Omron Sysmac Studio project OSU_Capstone_PI_Control (Sysmac Studio 1.47.0.64008, StandardProject)

# Controller new_Controller_0: NX1P2-9024DT1 version 1.40
Units and slaves: Unit 1 : NX-CIF101 (N1)
Task PrimaryTask (priority 4, period or condition 2000): Program0

VAR_GLOBAL
    Goto_Position : REAL := 0.0;
END_VAR
VAR_GLOBAL CONSTANT
    N1_Node_location_information : _sNXUNIT_ID := (NodeAdr := 65535, IPAdr := [5(16#FF)], UnitNo := 1, Path := [16#1, 16#0, 16#2, 16#0, 16#1, 59(16#0)], PathLength := 6);
END_VAR
VAR_GLOBAL
    DevicePort : _sDEVICE_PORT;
    trigger : BOOL;
    SendCfg : _sSERIAL_CFG;
    SendDat : ARRAY[0..49] OF BYTE;
    SendSiz : UINT;
    NX_SerialSend_FB_done : BOOL;
    NX_SerialSend_FB_busy : BOOL;
    NX_SerialSend_FB_err : BOOL;
    NX_SerialSend_FB_errID : WORD;
    trigger1 : BOOL;
    RecvCfg : _sSERIAL_CFG;
    RecvOption : _sSERIAL_RCV_OPTION;
    NX_SerialRcv_FB_done : BOOL;
    RecvDat : ARRAY[0..254] OF BYTE;
    NX_SerialRcv_FB_busy : BOOL;
    NX_SerialRcv_FB_err : BOOL;
    NX_SerialRcv_FB_errID : WORD;
    RecvSize : UINT;
    RecvStringDat : STRING[256];
    restarting : BOOL;
    N1_Ch1_Input_SID : USINT;  (* at IOBus://unit#1/Ch1 Input SID *)
    N1_Ch1_Output_SID_Response : USINT;  (* at IOBus://unit#1/Ch1 Output SID Response *)
    N1_Ch1_Input_Sub_Info : WORD;  (* at IOBus://unit#1/Ch1 Input Sub Info *)
    N1_Ch1_Receive_Command_Flag : BOOL;  (* at IOBus://unit#1/Ch1 Input Data Type/Ch1 Receive Command Flag *)
    N1_Ch1_Send_Command_Flag : BOOL;  (* at IOBus://unit#1/Ch1 Output Data Type/Ch1 Send Command Flag *)
    Pos_String : STRING[15];
    E001_Output_Data_1 : DINT;  (* at ECAT://node#1/Output Data 1 *)
    E001_READY : BOOL;  (* at ECAT://node#1/Sensor Head Status Signal1/READY *)
    E001_STABILITY : BOOL;  (* at ECAT://node#1/Sensor Head Status Signal2/STABILITY *)
END_VAR

PROGRAM Program0
VAR
    NX_SerialSend_FB : NX_SerialSend;
    NX_SerialRcv_FB : NX_SerialRcv;
    clear_trigger : BOOL;
    CmdStage : INT;
    CIFCmdCode : WORD;
    ExpectedOutputSIDResponse : USINT;
    Servo_On : BOOL;
    Reference : BOOL;
    Move_Axis : BOOL;
    Get_Info : BOOL;
    Abort_Send : BOOL;
    Reset_Error : BOOL;
    Pos_length : UINT;
    Last_positon : REAL;
    Auto : BOOL;
    Run : BOOL;
    Next_Move : TON;
    Next_Pos : BOOL;
    ZW_Real : REAL;
    ZW_Temp : REAL;
END_VAR
VAR_EXTERNAL
    DevicePort : _sDEVICE_PORT;
END_VAR
VAR_EXTERNAL CONSTANT
    N1_Node_location_information : _sNXUNIT_ID;
END_VAR
VAR_EXTERNAL
    trigger : BOOL;
    SendCfg : _sSERIAL_CFG;
    SendDat : ARRAY[0..49] OF BYTE;
    SendSiz : UINT;
    NX_SerialSend_FB_done : BOOL;
    NX_SerialSend_FB_busy : BOOL;
    NX_SerialSend_FB_err : BOOL;
    NX_SerialSend_FB_errID : WORD;
    trigger1 : BOOL;
    RecvCfg : _sSERIAL_CFG;
    RecvOption : _sSERIAL_RCV_OPTION;
    NX_SerialRcv_FB_done : BOOL;
    RecvDat : ARRAY[0..254] OF BYTE;
    NX_SerialRcv_FB_busy : BOOL;
    NX_SerialRcv_FB_err : BOOL;
    NX_SerialRcv_FB_errID : WORD;
    RecvSize : UINT;
    RecvStringDat : STRING[256];
    N1_Ch1_Input_SID : USINT;
    N1_Ch1_Output_SID_Response : USINT;
    restarting : BOOL;
    N1_Ch1_Send_Command_Flag : BOOL;
    N1_Ch1_Receive_Command_Flag : BOOL;
    N1_Ch1_Input_Sub_Info : WORD;
    Goto_Position : REAL;
    Pos_String : STRING[15];
    E001_STABILITY : BOOL;
    E001_READY : BOOL;
    E001_Output_Data_1 : DINT;
END_VAR
VAR
    _e1 : R_TRIG;
    _e2 : R_TRIG;
    _e3 : R_TRIG;
    _e4 : R_TRIG;
    _e5 : R_TRIG;
    _e6 : R_TRIG;
    _e7 : R_TRIG;
    _e8 : R_TRIG;
    _e9 : R_TRIG;
END_VAR

(* Section Serial_Setup: ladder, written here as Structured Text *)

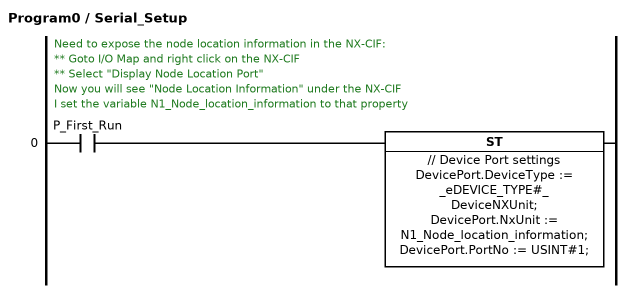
(* Rung 0: Need to expose the node location information in the NX-CIF: / ** Goto I/O Map and right click on the NX-CIF / ** Select "Display Node Location Port" / Now you will see "Node Location Information" under the NX-CIF / I set the variable N1_Node_location_information to that property *)
IF P_First_Run THEN
    // Device Port settings
    DevicePort.DeviceType := _eDEVICE_TYPE#_DeviceNXUnit;
    DevicePort.NxUnit := N1_Node_location_information;
    DevicePort.PortNo := USINT#1;
END_IF;

(* Section Serial_Send: ladder, written here as Structured Text *)

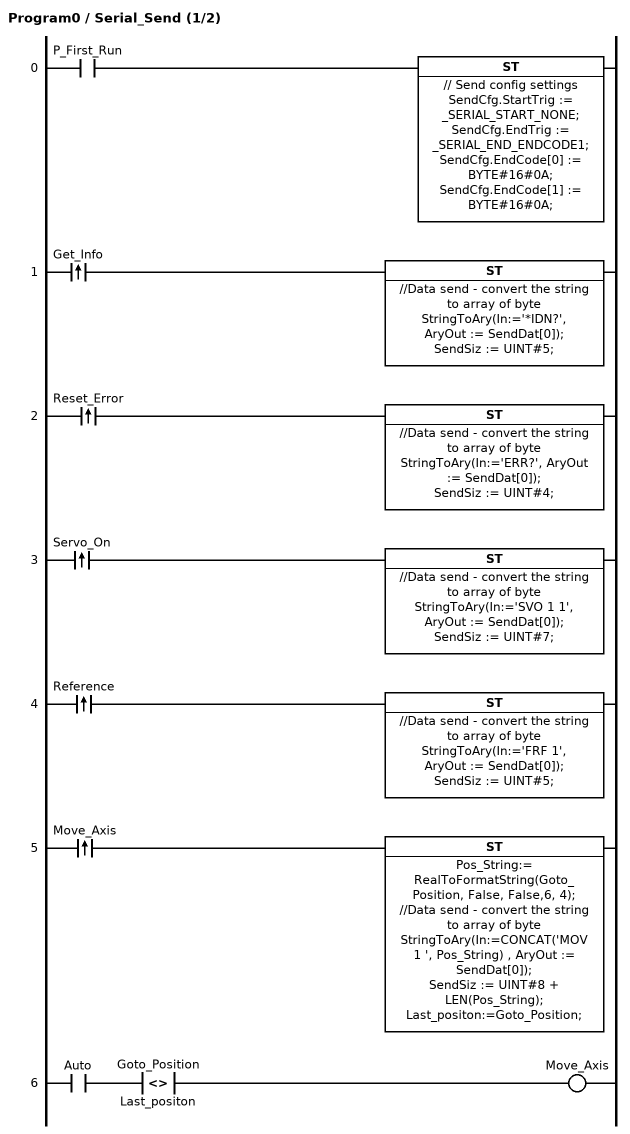
(* Rung 0 *)
IF P_First_Run THEN
    // Send config settings
    SendCfg.StartTrig := _SERIAL_START_NONE;
    SendCfg.EndTrig := _SERIAL_END_ENDCODE1;
    SendCfg.EndCode[0] := BYTE#16#0A;
    SendCfg.EndCode[1] := BYTE#16#0A;
END_IF;
(* Rung 1 *)
_e1(CLK := Get_Info);
IF _e1.Q THEN
    //Data send - convert the string to array of byte
    StringToAry(In:='*IDN?', AryOut := SendDat[0]);
    SendSiz := UINT#5;
END_IF;
(* Rung 2 *)
_e2(CLK := Reset_Error);
IF _e2.Q THEN
    //Data send - convert the string to array of byte
    StringToAry(In:='ERR?', AryOut := SendDat[0]);
    SendSiz := UINT#4;
END_IF;
(* Rung 3 *)
_e3(CLK := Servo_On);
IF _e3.Q THEN
    //Data send - convert the string to array of byte
    StringToAry(In:='SVO 1 1', AryOut := SendDat[0]);
    SendSiz := UINT#7;
END_IF;
(* Rung 4 *)
_e4(CLK := Reference);
IF _e4.Q THEN
    //Data send - convert the string to array of byte
    StringToAry(In:='FRF 1', AryOut := SendDat[0]);
    SendSiz := UINT#5;
END_IF;
(* Rung 5 *)
_e5(CLK := Move_Axis);
IF _e5.Q THEN
    Pos_String:= RealToFormatString(Goto_Position, False, False,6, 4);
    //Data send - convert the string to array of byte
    StringToAry(In:=CONCAT('MOV 1 ', Pos_String) , AryOut := SendDat[0]);
    SendSiz := UINT#8 + LEN(Pos_String);
    Last_positon:=Goto_Position;
END_IF;
(* Rung 6 *)
Move_Axis := Auto AND (Goto_Position <> Last_positon);

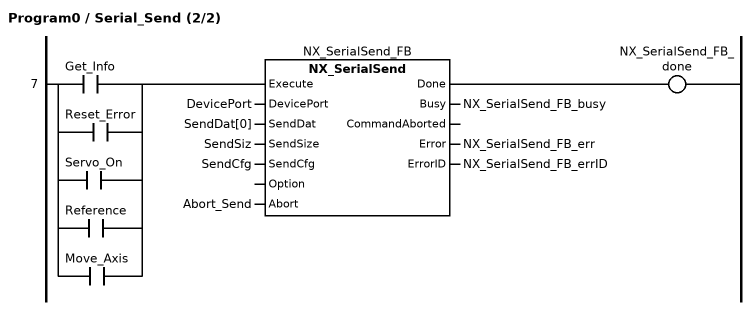
(* Rung 7 *)
NX_SerialSend_FB(Execute := Get_Info OR Reset_Error OR Servo_On OR Reference OR Move_Axis, DevicePort := DevicePort, SendDat := SendDat[0], SendSize := SendSiz, SendCfg := SendCfg, Abort := Abort_Send, Busy => NX_SerialSend_FB_busy, Error => NX_SerialSend_FB_err, ErrorID => NX_SerialSend_FB_errID);
NX_SerialSend_FB_done := NX_SerialSend_FB.Done;

(* Section Serial_Rec: ladder, written here as Structured Text *)

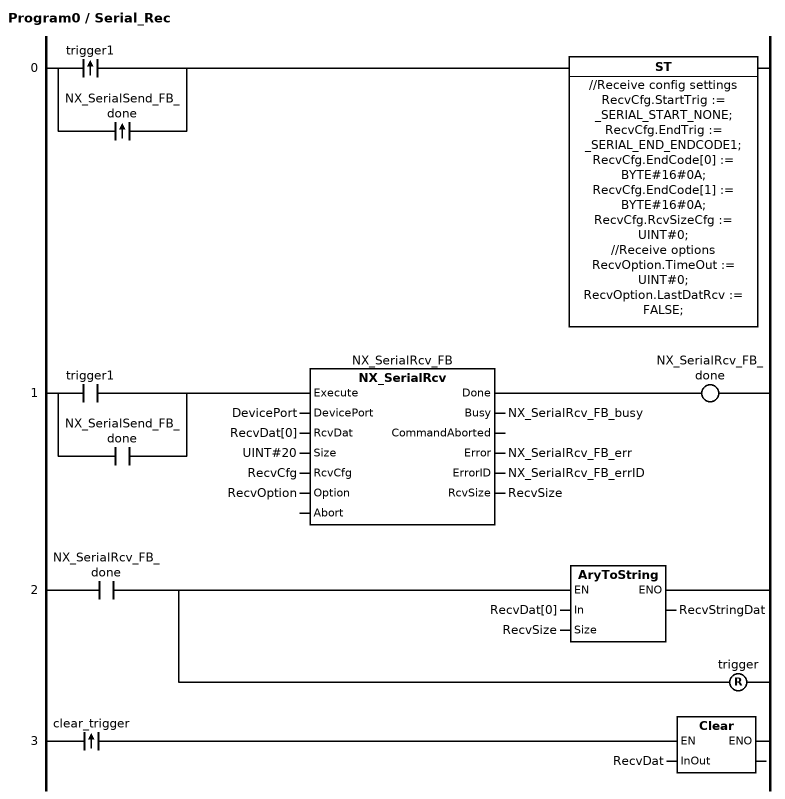
(* Rung 0 *)
_e6(CLK := trigger1);
_e7(CLK := NX_SerialSend_FB_done);
IF _e6.Q OR _e7.Q THEN
    //Receive config settings
    RecvCfg.StartTrig := _SERIAL_START_NONE;
    RecvCfg.EndTrig := _SERIAL_END_ENDCODE1;
    RecvCfg.EndCode[0] := BYTE#16#0A;
    RecvCfg.EndCode[1] := BYTE#16#0A;
    RecvCfg.RcvSizeCfg := UINT#0;
    //Receive options
    RecvOption.TimeOut := UINT#0;
    RecvOption.LastDatRcv := FALSE;
END_IF;
(* Rung 1 *)
NX_SerialRcv_FB(Execute := trigger1 OR NX_SerialSend_FB_done, DevicePort := DevicePort, RcvDat := RecvDat[0], Size := UINT#20, RcvCfg := RecvCfg, Option := RecvOption, Busy => NX_SerialRcv_FB_busy, Error => NX_SerialRcv_FB_err, ErrorID => NX_SerialRcv_FB_errID, RcvSize => RecvSize);
NX_SerialRcv_FB_done := NX_SerialRcv_FB.Done;
(* Rung 2 *)
IF NX_SerialRcv_FB_done THEN
    RecvStringDat := AryToString(In := RecvDat[0], Size := RecvSize);
    trigger := FALSE;
END_IF;
(* Rung 3 *)
_e8(CLK := clear_trigger);
IF _e8.Q THEN Clear(InOut := RecvDat); END_IF;

(* Section Auto: ladder, written here as Structured Text *)

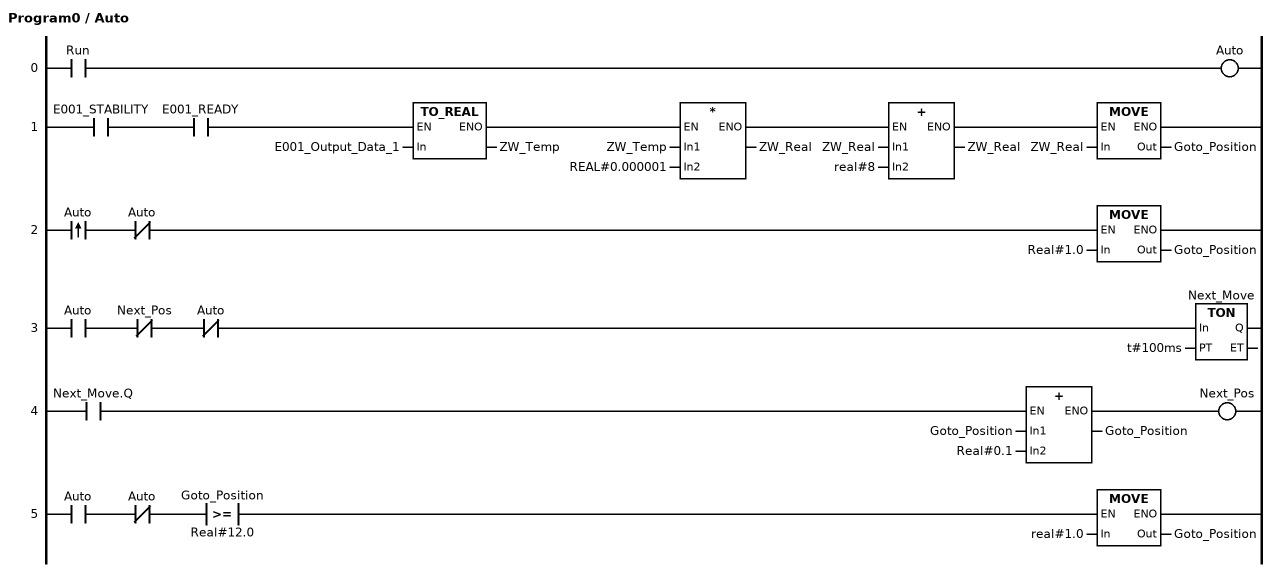
(* Rung 0 *)
Auto := Run;
(* Rung 1 *)
IF E001_STABILITY AND E001_READY THEN
    ZW_Temp := TO_REAL(In := E001_Output_Data_1);
    ZW_Real := ZW_Temp * REAL#0.000001;
    ZW_Real := ZW_Real + real#8;
    Goto_Position := ZW_Real;
END_IF;
(* Rung 2 *)
_e9(CLK := Auto);
IF _e9.Q AND NOT Auto THEN Goto_Position := Real#1.0; END_IF;
(* Rung 3 *)
Next_Move(In := Auto AND NOT Next_Pos AND NOT Auto, PT := t#100ms);
(* Rung 4 *)
IF Next_Move.Q THEN Goto_Position := Goto_Position + Real#0.1; END_IF;
Next_Pos := Next_Move.Q;
(* Rung 5 *)
IF Auto AND NOT Auto AND (Goto_Position >= Real#12.0) THEN Goto_Position := real#1.0; END_IF;
END_PROGRAM